ABB RobotStudio station: material handling achu 4 3 24_1.rsstn

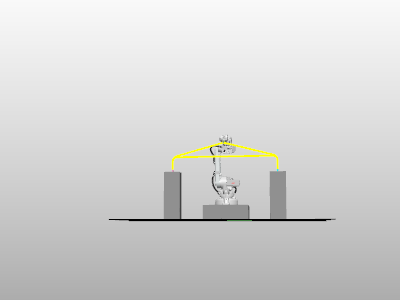
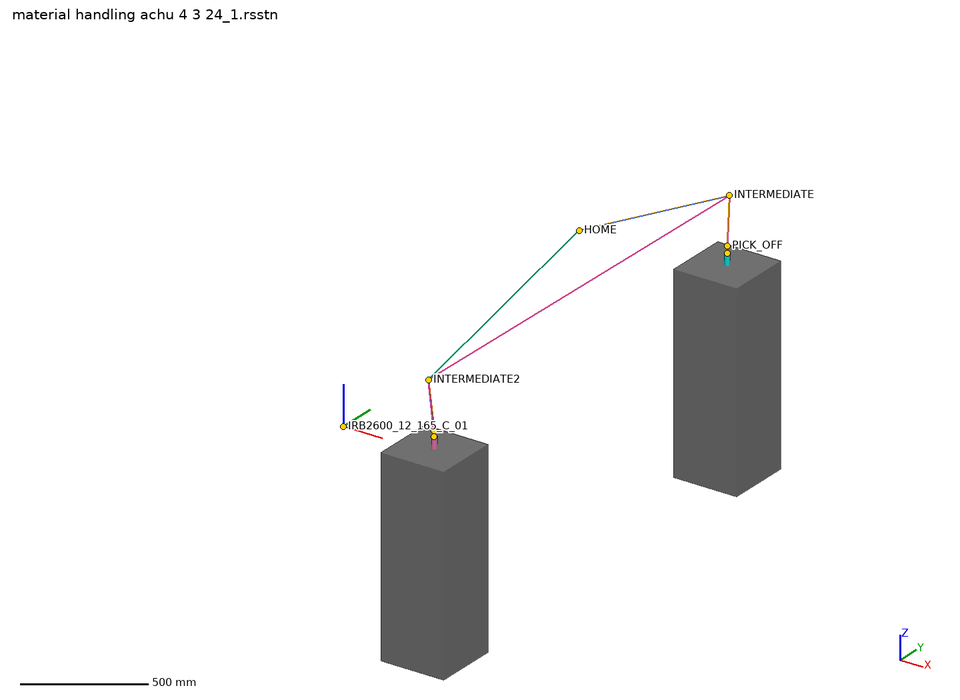
[picture v1: parts stored in the station drawn from their meshes, with robot base, taught points and paths (robot models come from the ABB library and are not in the file)]
Station Station (saved by RobotStudio 22.3.10141.1)
Controller Controller22, task T_ROB1: task frame (RAPID world) sits at (0, 0, 300) mm in the station
Controller Controller22
  mechanical unit ROB_1: IRB2600_12_165_C_01, 6 joints, base frame (0, 0, 0) mm
Layout (positions relative to the parent item):
  - concrete [part, from Libraries\concrete.rslib] at (-450, -450, 0) mm
  - IRB2600_12_165_C_01 [mechanism, from %ABB.RobotStudio.Models.IRB2600%\IRB2600_12_165_C_01.rslib] at (0, 0, 300) mm; joint values [0, 0, 0, 0, 0.5236, 0] (rad or m)
  - SmartComponent_1 [smart component] at (1018.61, 0, 1517.5) mm, rotated rx 180 ry 60 rz 180 deg
      signals: DI attach
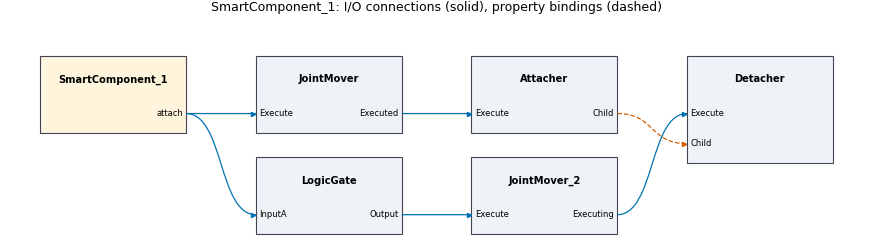
      connections:
        SmartComponent_1.attach -> JointMover.Execute
        JointMover.Executed -> Attacher.Execute
        SmartComponent_1.attach -> LogicGate.InputA
        LogicGate.Output -> JointMover_2.Execute
        JointMover_2.Executing -> Detacher.Execute
        Attacher.Child => Detacher.Child
    - Smart_Gripper_Servo_Fingers [mechanism, from Tools\ABB_Smart_Gripper_Servo_Fingers.rslib] at (0, 0, 0) mm; joint values [0.025] (rad or m)
    - JointMover [smart component, from Components\JointMover.rslib]
        properties: Mechanism=Smart_Gripper_Servo_Fingers; Relative=false; Duration=0; J1=0.023
    - JointMover_2 [smart component, from Components\JointMover.rslib]
        properties: Mechanism=Smart_Gripper_Servo_Fingers; Relative=false; Duration=0; J1=0.025
    - Attacher [smart component, from Components\Attacher.rslib]
        properties: Parent=Smart_Gripper_Servo_Fingers; Flange=0; Child=object; Mount=false; Offset=[0 0 0]; Orientation=[0 0 0]
    - LogicGate [smart component, from Components\LogicGate.rslib]
        properties: Operator=NOT; Delay=0
    - Detacher [smart component, from Components\Detacher.rslib]
        properties: Child=object; KeepPosition=true
  - table_1 [part] at (955.3, 870.39, 0) mm, size 300 x 300 x 900 mm
  - table_2 [part] at (955.3, -1114.68, 0) mm, size 300 x 300 x 900 mm
  - object [part] at (1105.3, 1020.39, 900) mm, size 24 x 23.9 x 50 mm
  - object_3 [part] at (1105.3, -964.68, 900) mm, size 24 x 23.9 x 50 mm
Attachment: SmartComponent_1 is attached to IRB2600_12_165_C_01 / Link6
Station logic (signal -> signal, property => property):
  Controller22.attach -> SmartComponent_1.attach
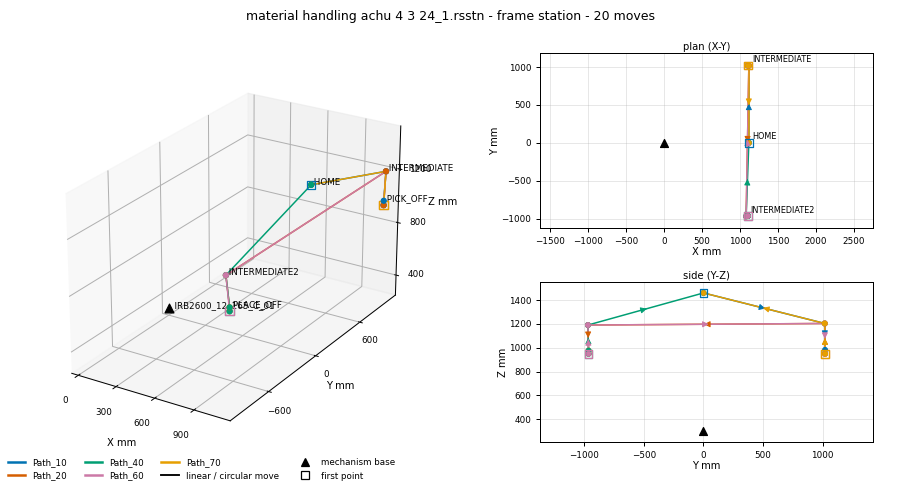
[picture p0: tool path of material handling achu 4 3 24_1.rsstn in frame station, 20 of 20 moves have a stored position in this frame; points joined in program order, loops and branches not executed]
Targets, tools, work objects and paths stored in the station, written as RAPID:
! task T_ROB1
MODULE CalibData
  PERS tooldata Servo:=[TRUE,[[0,0,114.2],[1,0,0,0]],[0.215,[8.7,12.3,49.2],[1,0,0,0],0.00021,0.00024,0.00009]];
ENDMODULE

! task T_ROB1
MODULE Module1
  CONST robtarget HOME:=[[1117.512260434,0,1160.4],[0.5,0,0.866025404,0],[-1,0,-1,0],[9E+09,9E+09,9E+09,9E+09,9E+09,9E+09]];
  CONST robtarget INTERMEDIATE:=[[1117.511980946,1017.932050718,904.191201819],[0.500000012,-0.000000076,0.866025397,-0.00000001],[0,-1,0,0],[9E+09,9E+09,9E+09,9E+09,9E+09,9E+09]];
  CONST robtarget PICK:=[[1105.303020676,1020.390036577,650.000489152],[0.013999954,0.790796768,-0.611666722,-0.017558305],[0,0,-1,0],[9E+09,9E+09,9E+09,9E+09,9E+09,9E+09]];
  CONST robtarget PICK_OFF:=[[1105.303031261,1020.390043529,682.542153466],[0.013999902,0.790796807,-0.611666673,-0.017558292],[0,0,-1,0],[9E+09,9E+09,9E+09,9E+09,9E+09,9E+09]];
  CONST robtarget INTERMEDIATE2:=[[1081.886978598,-969.801506265,891.044657892],[0.013999873,0.790796514,-0.611667052,-0.017558331],[-1,-1,-2,0],[9E+09,9E+09,9E+09,9E+09,9E+09,9E+09]];
  CONST robtarget PLACE:=[[1105.303042071,-964.684458552,650.000520506],[0.013999871,0.790796526,-0.611667034,-0.017558383],[-1,-1,-2,0],[9E+09,9E+09,9E+09,9E+09,9E+09,9E+09]];
  CONST robtarget PLACE_OFF:=[[1105.303050199,-964.684465643,676.304740266],[0.013999872,0.790796537,-0.611667021,-0.017558352],[-1,-1,-2,0],[9E+09,9E+09,9E+09,9E+09,9E+09,9E+09]];
  PROC Path_10()
    MoveL HOME,v1000,z100,Servo\WObj:=wobj0;
    MoveL INTERMEDIATE,v1000,z100,Servo\WObj:=wobj0;
    MoveL PICK_OFF,v1000,z100,Servo\WObj:=wobj0;
    MoveL PICK,v1000,z100,Servo\WObj:=wobj0;
    WaitTime 1;
    SetDO attach,1;
    WaitTime 1;
  ENDPROC
  PROC Path_20()
    MoveL PICK,v1000,z100,Servo\WObj:=wobj0;
    MoveL INTERMEDIATE,v1000,z100,Servo\WObj:=wobj0;
    MoveL INTERMEDIATE2,v1000,z100,Servo\WObj:=wobj0;
    MoveL PLACE_OFF,v1000,z100,Servo\WObj:=wobj0;
    MoveL PLACE,v1000,z100,Servo\WObj:=wobj0;
    WaitTime 1;
    SetDO attach,0;
    WaitTime 1;
  ENDPROC
  PROC Path_40()
    MoveL PLACE,v1000,z100,Servo\WObj:=wobj0;
    MoveL PLACE_OFF,v1000,z100,Servo\WObj:=wobj0;
    MoveL INTERMEDIATE2,v1000,z100,Servo\WObj:=wobj0;
    MoveL HOME,v1000,z100,Servo\WObj:=wobj0;
  ENDPROC
  PROC main()
  ENDPROC
  PROC Path_50()
    Path_10;
    Path_20;
    Path_40;
    Path_60;
    Path_70;
  ENDPROC
  PROC Path_60()
    MoveL PLACE,v1000,z100,Servo\WObj:=wobj0;
    WaitTime 1;
    SetDO attach,1;
    WaitTime 1;
    MoveL INTERMEDIATE2,v1000,z100,Servo\WObj:=wobj0;
    MoveL INTERMEDIATE,v1000,z100,Servo\WObj:=wobj0;
    MoveL PICK,v1000,z100,Servo\WObj:=wobj0;
    WaitTime 1;
    SetDO attach,0;
    WaitTime 1;
  ENDPROC
  PROC Path_70()
    MoveL PICK,v1000,z100,Servo\WObj:=wobj0;
    MoveL INTERMEDIATE,v1000,z100,Servo\WObj:=wobj0;
    MoveL HOME,v1000,z100,Servo\WObj:=wobj0;
  ENDPROC
ENDMODULE

